PROGRAM MAIN
VAR
	//To attach variables to IO modules, it is needed to use "AT",
	// Inputs - I, Output - Q 
	bStart AT %I* 	: BOOL; 		// start button
	bLamp AT %Q*	: BOOL;			// Lamp 
	
	// Local variables without connecting to IO
	bStatus 		: BOOL;
	
END_VAR


// Switch on the lamp with push button in visualization.
bLamp := bStart;

END_PROGRAM

(* stored: Version 1.1.0.1, ProductVersion 3.1.4022.16
   POU MAIN: Id {57ff0dc6-447c-4b99-9c33-6a346549c215}, SpecialFunc None *)
